FUNCTION_BLOCK clock_gen
  (* Standard: 61499-2 *)
  (* Version 0,1, 2015-00-09, Th?o, PC_THEO *)
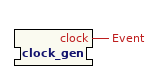
  EVENT_OUTPUT
    clock;
  END_EVENT
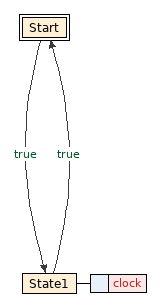
  EC_STATES
    Start;
    State1 : -> clock;
  END_STATES
  EC_TRANSITIONS
    Start TO State1 := true;
    State1 TO Start := true;
  END_TRANSITIONS
END_FUNCTION_BLOCK
